ABB RobotStudio station: MTRN4230.rsstn

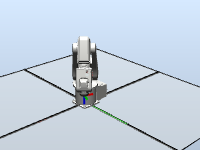
Station Station (saved by RobotStudio format 3)
Controller MTRN4230
  mechanical unit ROB_1: IRB120_3_58__01, 6 joints, base frame (0, 0, 0) mm
Layout (positions relative to the parent item):
  - IRB120_3_58__01 [mechanism, from Robots\IRB120_3_58_G_01.rslib] at (0, 0, 0) mm; joint values [0.8326, 0.4284, 0.7299, 0.0018, 0.4128, 1.1804] (rad or m)
